PROGRAM MAIN
VAR
	bDoorC AT%Q* : BOOL;
	bDoorO AT%Q* : BOOL;
	bVentil AT%I* : BOOL;
	
	fbTestMaschinentuer : FB_TestMaschinentuer;
END_VAR


fbTestMaschinentuer(bVentil:= bVentil ,
 					bDoorC=> bDoorC , 
					bDoorO=> bDoorO);

END_PROGRAM

(* stored: Version 1.1.0.1, ProductVersion 3.1.4024.15
   POU MAIN: Id {289bbdbb-ad67-4d57-86ad-3245f2cb5119}, SpecialFunc None *)
